// TwinCAT 3 PLC project API
// ProgramVersion: 3.1.4020.4
// libraries:
//   Tc2_MC2, * (Beckhoff Automation GmbH)
//   Tc2_Standard, * (Beckhoff Automation GmbH)
//   Tc2_System, * (Beckhoff Automation GmbH)
//   Tc3_Module, * (Beckhoff Automation GmbH)
// project tree:
//   DUTs/ ST_GenericStatus.TcDUT, ST_IO.TcDUT, ST_MachineParam.TcDUT, ST_Out.TcDUT, ST_Param.TcDUT, ST_RecipeParam.TcDUT, ST_Status.TcDUT
//   GVLs/ GVL.TcGVL
//   / PlcTask.TcTTO
//   POUs/ FB_Btn.TcPOU, FB_BtnHmiAutoResetType.TcPOU, FB_CycleAuto.TcPOU, FB_CycleInit.TcPOU, FB_CycleMain.TcPOU, FB_CycleMan.TcPOU, FB_Moteur.TcPOU, FB_Station.TcPOU, MAIN.TcPOU
// real-time tasks:
//   TASK PlcTask: cycle T#10ms, priority 20, ADS port 350
// motion (NC):
//   TASK NC-Task 1 SAF: cycle T#2ms, priority 4, ADS port 501
//   TASK NC-Task 1 SVB: cycle T#10ms, priority 8, ADS port 511
//   AXIS Axe Z (id 1)
//     OtherSettings: AllowMotionCmdToSlave=true
//     encoder EncType=1
//     drive DrvType=5
//     controller CtrType=1
//       CtrPara: PriorControlFactor=1
//         Observer: BandWidth=20
// variable links:
//   API/API Instance <-> NC-Task 1 SAF/Axes/Axe Z
//     PlcTask Inputs/GVL.axeX.NcToPlc <-> Outputs/ToPlc
//     PlcTask Outputs/GVL.axeX.PlcToNc <-> Inputs/FromPlc

CONFIGURATION API
    RESOURCE PLC ON TwinCAT3
        TASK PlcTask(INTERVAL := T#10ms, PRIORITY := 20);
        PROGRAM MAIN WITH PlcTask : MAIN;
    END_RESOURCE
END_CONFIGURATION

// ---- DUTs/ST_GenericStatus.TcDUT
TYPE ST_GenericStatus :
STRUCT
	(*-------------------------------------------------------------------------------------------------
		xuton du panel HMI
	-------------------------------------------------------------------------------------------------*)
	(*mode actif plc to HMI*)
	xModeInit					:BOOL; (*selection du mode prise origine machine type flanc*)
	

	xModeAuto				:BOOL; (*selection du mode automatique type flanc*)
	xModeMan				:BOOL; (*selection du mode manuel type flanc*)
	xModeStep				:BOOL; (*selection du mode pas à pas type flanc*)
	
	xWaitStartNextStep:BOOL;

	iNcStatus				:DINT;					(*status NC*)
	iOverride:DINT;
	(*-------------------------------------------------------------------------------------------------
		Machine global state
	-------------------------------------------------------------------------------------------------*)

	(*boReadyForPower			: BOOL;					(* Condition machine prête pour faire un power on des axes*)*)
	xInitOk:BOOL;


	xPowerOff:BOOL;(*"POWER OFF": IF motor power AND pneumatic are "OFF" (Emergency stop)*)

	xPowering:BOOL;(*"POWERING": Transition mode*)

	xPowerOn:BOOL;(*"POWER ON": Motor power "ON", pneumatic "ON"*)

	xInitializing:BOOL;(*"INITIALISING": Transition mode, INIT cycle*)

	xReady:BOOL;(*"READY": Ready FOR AUTO mode Green*)

	xRunning:BOOL;(*"RUNNING": running in AUTO mode*)

	xStoping:BOOL;(*"STOPPING": Normally stopping  in AUTO mode*)

	xReseting:BOOL;(*"RESETING": Reset cycle operation, can be DO in every situation AND mode*)

	(*Status light*)
	byStatusLight:BYTE; (*bit0=1 red light, bit1=1 red light blink, bit2=1 yelow, bit3=1 yelow blink, bit4=1 green, bit5=1 green blink*)

END_STRUCT
END_TYPE

// ---- DUTs/ST_IO.TcDUT
TYPE ST_IO :
STRUCT
	stOut: ST_Out;
END_STRUCT
END_TYPE

// ---- DUTs/ST_MachineParam.TcDUT
TYPE ST_MachineParam :
STRUCT
	
END_STRUCT
END_TYPE

// ---- DUTs/ST_Out.TcDUT
TYPE ST_Out :
STRUCT
	xMotEnable: BOOL;
	xMotPosBasse: BOOL;
	xMotPosHaute: BOOL;
END_STRUCT
END_TYPE

// ---- DUTs/ST_Param.TcDUT
TYPE ST_Param :
STRUCT
	
	(*NOVRAM (Non-Volatile Random Access Memory) persistent variables *)
	(*Parameters*)
	stStatus		:ST_Status;	(*Machine global status structure ~(OPC :1:)*)
	stMachine		:ST_MachineParam ;	(*Machine parameters structure editing from HMI ~(OPC :1:)*)
	stRecipe		:ST_RecipeParam;	(*Recipe parameters structure editing from HMI ~(OPC :1:)*)
	//stReporting		:ST_Reporting;
	

END_STRUCT
END_TYPE

// ---- DUTs/ST_RecipeParam.TcDUT
TYPE ST_RecipeParam :
STRUCT

	(*Paramètres production*)
	lrPositionBasse: LREAL;
	lrVitesse: LREAL;
	
END_STRUCT
END_TYPE

// ---- DUTs/ST_Status.TcDUT
TYPE ST_Status :
STRUCT
	(*Common*)
	stCommon:ST_GenericStatus;	(*Common*)

	(*Activation from HMI*)
	inJogSelectCylinder:INT;(**)
	inJogSelectMotor: INT;
	iNiveauUtilisateur:INT;
	sUserName:STRING[100]:='';//user name from HMI
	
	iCounterPiecesProduites: INT;                             (*Nombre de pièces produites (=nombre de pièces triées)*)
	iCounterPiecesBonnes: INT;
	iCounterPiecesMauvaises: INT;
	iCounterLaser:DINT;//compteur de cycle laser limite à 4'000'000
	diCounterError:DINT;
	//sMessageHmi: STRING(200);
	sMessageHmiStatus: STRING(50);	
	sBatchNo:STRING[50];
	
	//indique le niveau, vrai si plus gand ou égale
	xNiveau1:BOOL;
	xNiveau2:BOOL;
	xNiveau3:BOOL;
	xNiveau4:BOOL;
	
	lrPositionMoteur: LREAL;
	
END_STRUCT
END_TYPE

// ---- GVLs/GVL.TcGVL
VAR_GLOBAL
fbStation		:FB_Station;(*Function Block for  station*)
stIO: ST_IO;
axeX: AXIS_REF;
END_VAR

VAR_GLOBAL PERSISTENT
stParam:ST_Param;//Basis structure with all parameters and status
END_VAR

// ---- POUs/MAIN.TcPOU
PROGRAM MAIN
VAR
END_VAR

fbStation();

GVL.stParam.stStatus.lrPositionMoteur:=GVL.axeX.NcToPlc.ActPos;

GVL.stIO.stOut.xMotPosBasse:=GVL.axeX.NcToPlc.ActPos<=GVL.stParam.stRecipe.lrPositionBasse+0.01;

GVL.stIO.stOut.xMotPosHaute:=GVL.axeX.NcToPlc.ActPos>=-0.01;

END_PROGRAM

// ---- POUs/FB_Station.TcPOU
FUNCTION_BLOCK FB_Station
VAR_INPUT
	(*Objets*)
	
	
	(*Function block for cycle*)
	fbCycleMain:FB_CycleMain;
	fbCycleInit:FB_CycleInit;
	fbCycleMan:FB_CycleMan;
	fbCycleAuto:FB_CycleAuto;
	
	fbAxeX: FB_Moteur;
	
	
	(*Function blockfor small HMI button*)
	fbBtn:FB_Btn;	(*station Input and ouput*)

	(*Error management*)
//	fbErrorAdmin		:FB_ErrorAdmin;	(*FUNCTION block for error administration  *)
	
	
	
END_VAR
VAR_OUTPUT

END_VAR
VAR
	
END_VAR

//fbErrorAdmin.mResetIndex();
(************************************************************************************)
(*							Refresh cycle			 *)
(************************************************************************************)
ACT_Cycle();
ACT_Refresh();
//fbIO();
fbBtn();

fbCycleMain();

ACT_ActionActionneur();

ACTION ACT_ActionActionneur:
fbAxeX.fbHome.Execute:=fbStation.fbCycleInit.iStep=100;
fbAxeX.fbReset.Execute:=fbStation.fbCycleMain.iStep=820;
fbAxeX.fbMoveAbsolute.Execute:=fbStation.fbCycleAuto.iStep=200 OR fbStation.fbCycleAuto.iStep=300;
fbAxeX(fbAxe:=GVL.axeX);
fbAxeX.fbPower.Enable:=GVL.stIO.stOut.xMotEnable;
fbAxeX.fbPower.Enable_Negative:=TRUE;
fbAxeX.fbPower.Enable_Positive:=TRUE;
END_ACTION

ACTION ACT_Cycle:


(*Start cycle in mode*)
fbCycleInit.xStart:=fbStation.fbCycleMain.iStep=150;

fbCycleMan.xStart:=fbStation.fbCycleMain.iStep=200;

fbCycleAuto.xStart:=fbStation.fbCycleMain.iStep=305;
//fbCycleAuto.xStopCmdPin:=fbStation.fbCycleMain.iStep=390  OR fbStation.fbCycleMain.iStep=800;


fbCycleInit( );
fbCycleMan(  );
fbCycleAuto( );
END_ACTION

ACTION ACT_Refresh:
	


	(*"POWER OFF": IF motor power AND pneumatic are "OFF" (Emergency stop)
	IF this machine is selected AND power Off, it correspond TO an alarm. Red is OK.
	IF this machine isn't selected and power Off, it must be white.*)
	//stParam.stStatus.stCommon.xPowerOff:=fbStation.fbIO.In.IxEstopBtnOnly;

	(*"POWERING": Transition mode
	IF the machines are powering but without alarms OR warnings, they can blink in light blue.
	IF the machines are powering but with warning, they can blink in yellow.
	IF the machines are powering but with alarms, they can blink in red.*)
	stParam.stStatus.stCommon.xPowering:=FALSE;

	(*"POWER ON": Motor power "ON", pneumatic "ON"
	IF the machines are power On but without alarms OR warnings, they can be light blue.
	IF the machines are power On but with warning, they can be yellow.
	IF the machines are power On but with alarms, they can be red.*)
	//stParam.stStatus.stCommon.xPowerOn:=NOT fbStation.fbIO.In.IxEstopBtnOnly;

	(*"INITIALISING": Transition mode, INIT cycle
	IF the machines are initializing but without alarms OR warnings, they can blink in green.
	IF the machines are initializing but with warning, they can blink in yellow.
	IF the machines are initializing but with alarms, they can blink in red.*)
	stParam.stStatus.stCommon.xInitializing:=fbStation.fbCycleMain.iStep>100 AND fbStation.fbCycleMain.iStep<199;

	

	(*"RUNNING": running in AUTO mode
	IF the machines are running but without alarms OR warnings, they can blink in green.
	IF the machines are running but with warning, they can blink in yellow.
	IF the machines are running but with alarms, they can blink in red (NOT possible).*)
	stParam.stStatus.stCommon.xRunning:= fbStation.fbCycleAuto.xBusy
										OR fbStation.fbCycleInit.xBusy OR fbStation.fbCycleMan.iStep>5;
										
	stParam.stStatus.stCommon.xReady:=NOT stParam.stStatus.stCommon.xRunning
								 AND stParam.stStatus.stCommon.xPowerOn
								AND stParam.stStatus.iNiveauUtilisateur>0;
								 
	(*"STOPPING": Normally stopping  in AUTO mode
	IF the machines are stopping but without alarms OR warnings, they can blink in green.
	IF the machines are stopping but with warning, they can blink in yellow.
	IF the machines are stopping but with alarms, they can blink in red (NOT possible).*)
	stParam.stStatus.stCommon.xStoping:=fbStation.fbCycleMain.iStep=390  OR fbStation.fbCycleMain.iStep=800;

	(*"RESETING": Reset cycle operation, can be DO in every situation AND mode
	IF the machines are stopping but without alarms OR warnings, they can blink in green.
	IF the machines are stopping but with warning, they can blink in yellow.
	IF the machines are stopping but with alarms, they can blink in red.*)
	stParam.stStatus.stCommon.xReseting:=fbStation.fbCycleMain.xReseting;


IF stParam.stStatus.stCommon.xRunning
		THEN
		 IF stParam.stStatus.stCommon.xWaitStartNextStep 
			 THEN
			 	stParam.stStatus.sMessageHmiStatus:='SETP BY STEP';
			 ELSE
				stParam.stStatus.sMessageHmiStatus:='RUN';
		END_IF
		ELSE
			stParam.stStatus.sMessageHmiStatus:='READY';
END_IF

stParam.stStatus.xNiveau1:=stParam.stStatus.iNiveauUtilisateur>0;
stParam.stStatus.xNiveau2:=stParam.stStatus.iNiveauUtilisateur>1;
stParam.stStatus.xNiveau3:=stParam.stStatus.iNiveauUtilisateur>2;
stParam.stStatus.xNiveau4:=stParam.stStatus.iNiveauUtilisateur>3;

//Visibilité/invisibilité des boutons de quittance:
(*
stParam.stStatus.xBtnQuittanceBal1Visible:=	fbStation.fbCycleBalance1.iStep=802
												OR fbStation.fbCycleBalance1.iStep=842
												OR fbStation.fbCycleVerifEtatStation.iStep=160;
stParam.stStatus.xBtnQuittanceBal2Visible:=	fbStation.fbCycleBalance2.iStep=804	
												OR fbStation.fbCycleBalance2.iStep=844
												OR fbStation.fbCycleVerifEtatStation.iStep=210;
stParam.stStatus.xBtnQuittanceUsiVisible:=	fbStation.fbCycleUsinage.iStep=812
												OR fbStation.fbCycleVerifEtatStation.iStep=260;
*)
END_ACTION

END_FUNCTION_BLOCK

// ---- POUs/FB_CycleMain.TcPOU
FUNCTION_BLOCK FB_CycleMain
(**)
VAR_INPUT

END_VAR
VAR_OUTPUT
	xBusy				:BOOL;(*Busy output*)
	xReseting:BOOL;(*reseting mode*)
	xReadyForChangingMode:bool;
	xEStopOut:BOOL;
END_VAR
VAR_IN_OUT
END_VAR
VAR
	iStep			: INT:=0;		(* cycle step *)
	inOldStep			:INT:=0;
	fbTrigStart			: R_Trig;	(*Trigger for start*)
	
	xMemCycleAutoRun:BOOL;
	
	fbTimer:TON;
	fbTimerResetAuto:ton;
END_VAR



ACT_ChangingMode();


IF fbStation.fbBtn.HmiReset.xRisingEdge AND iStep<800
	THEN
		iStep:=800;
END_IF

CASE  iStep OF

	(********************************************************************************************************************************************************)
	(*Plc Start*)
	(********************************************************************************************************************************************************)
	0:	(*Init*)
		iStep:=50;
	
		
	(*Select mode*)
	50:(*Wait end of cycle man init auto*)
		//boEndOfProdPout:=FALSE;
		IF xReadyForChangingMode
			THEN
				iStep:=55;
		END_IF
		
	55:	(*Changing mode from HMI*)
		(*Select  Mode*)
		IF  stParam.stStatus.stCommon.xModeInit
			THEN
				iStep:=100; (*Init mode*)
		END_IF
		IF stParam.stStatus.stCommon.xModeMan 
			THEN
				iStep:=200; (*Manual mode*)
		END_IF
		IF stParam.stStatus.stCommon.xModeAuto
			THEN
					iStep:=300;(*Auto mode*)
		END_IF

	(************************************************************************************)
	(*							INIT mode						 *)
	(************************************************************************************)
	(*Wait for start cycle or changing mode*)
	100:
		IF NOT stParam.stStatus.stCommon.xModeInit
			THEN
				iStep:=50;(*select mode*)
			ELSE
				(*Start init*)
				IF (fbStation.fbBtn.HmiStart.xRisingEdge)
					THEN
						iStep:=150;
				END_IF
		END_IF

	150:(*Exit on normal end*)
		IF fbStation.fbCycleInit.xDone
			THEN
				iStep:=190;
		END_IF
		(*Exit on reset*);
		(*Exit with error level 2*)
	(*End of INIT mode*)
	190:
		//changement de mode automatique AUTO
		iStep:=50;

	(************************************************************************************)
	(*							MAN mode						 *)
	(************************************************************************************)
	(*changing mode*)
	200:
		IF NOT stParam.stStatus.stCommon.xModeMan 
			THEN
				(*select mode*)
				iStep:=290;
		END_IF
	290:(*	stParam.stStatus.dsMotPortiqueM1.xKillMotor:=FALSE;
		stParam.stStatus.dsMotPortiqueM2.xKillMotor:=FALSE;
		stParam.stStatus.dsMotPump.xKillMotor:=FALSE;*)
		IF NOT fbStation.fbCycleMan.xBusy
				THEN
					iStep:=50;
		END_IF
		

	(************************************************************************************)
	(*							AUTO mode						 *)
	(************************************************************************************)
	(*changing mode*)
	300:
		IF NOT stParam.stStatus.stCommon.xModeAuto
			THEN
				iStep:=50;(*select mode*)
			ELSE
				//Start cycle auto normal
				IF (fbStation.fbBtn.HmiStart.xRisingEdge)
					THEN
						iStep:=305;
				END_IF
		END_IF
	
	305: IF NOT fbStation.fbCycleAuto.xDone
		THEN
			iStep:=310;
	END_IF	
		
	(*Control*)
	310:IF fbStation.fbCycleAuto.xDone
		THEN
			GVL.stParam.stStatus.iCounterPiecesProduites:=GVL.stParam.stStatus.iCounterPiecesProduites+1;
			iStep:=300;
	END_IF

	(************************************************************************************)
	(*							Resetting mode					 *)
	(************************************************************************************)
	800:(*IF NOT fbStation.fbCycleAuto.xBusy OR fbTimerResetAuto.Q
			THEN
				iStep:=805;
		END_IF*)
		fbStation.fbCycleAuto.xReset:=TRUE;
		fbStation.fbCycleInit.xReset:=TRUE;
		fbStation.fbCycleMan.xReset:=TRUE;
		GVL.stIO.stOut.xMotEnable:=FALSE;
		iStep:=810;
		
	
	810:IF NOT fbStation.fbCycleInit.xBusy
		AND NOT fbStation.fbCycleMan.xBusy
		AND NOT fbStation.fbCycleAuto.xBusy
		THEN
			iStep:=820;
		END_IF
		
	820: IF fbStation.fbAxeX.fbReset.Done
		 THEN
		 	iStep:=830;
	END_IF
	
	830: GVL.stIO.stOut.xMotEnable:=TRUE;
		iStep:=50;

END_CASE

(********************************************************************************************************************************************************)
(*Special Interrupt*)
(********************************************************************************************************************************************************)




fbTimer(IN:=iStep=20 OR iStep=807 OR iStep=809 OR iStep=841 );
fbTimerResetAuto(IN:=iStep=800,pt:=T#1000MS);


xBusy:=(iStep<>0);
xReseting:=(iStep>799 AND iStep<900);



xReadyForChangingMode:= (iStep=100 OR iStep=200 OR iStep=300 OR iStep=50 OR iStep=55)
			AND NOT fbStation.fbCycleInit.xBusy
			AND NOT fbStation.fbCycleAuto.xBusy;

xEStopOut:= (iStep>899);


(********************************************************************************************************************************************************)
(*Status settings*)
(********************************************************************************************************************************************************)

xBusy:=(iStep<>0);
xReseting:=(iStep>799 AND iStep<900);

ACTION ACT_ChangingMode:
(*********************************************************************************)
(*			Changing mode														 *)
(*********************************************************************************)
IF (fbStation.fbBtn.Init.xRisingEdge 
	) 
	AND xReadyForChangingMode 
	THEN
		stParam.stStatus.stCommon.xModeInit:=TRUE;
		stParam.stStatus.stCommon.xModeAuto:=FALSE;
		stParam.stStatus.stCommon.xModeMan:=FALSE;
END_IF

IF fbStation.fbBtn.Auto.xRisingEdge 
	AND xReadyForChangingMode
 OR iStep=190 AND stParam.stStatus.stCommon.xInitOk
	THEN
		stParam.stStatus.stCommon.xModeInit:=FALSE;
		stParam.stStatus.stCommon.xModeAuto:=TRUE;
		stParam.stStatus.stCommon.xModeMan:=FALSE;
END_IF

IF fbStation.fbBtn.Man.xRisingEdge AND xReadyForChangingMode
	THEN
		stParam.stStatus.stCommon.xModeInit:=FALSE;
		stParam.stStatus.stCommon.xModeAuto:=TRUE;
		stParam.stStatus.stCommon.xModeMan:=FALSE;
END_IF
END_ACTION

ACTION ACT_ForceInitAllAxe:
stParam.stStatus.stCommon.xInitOk:=FALSE;
END_ACTION

END_FUNCTION_BLOCK

// ---- POUs/FB_CycleInit.TcPOU
(**********************************************************************************************************************************************************************
*{He-Arc}  {Hôtle de ville 7}   {2400 Le Locle}       Phone: ++ 0041 (0)32 930 13 13     Fax: ++ 0041 (0)32 930 13 14         Email: ingenierie@he-arc.ch
*=======================================================================================================================
* {Give the complete list of every blocks for a source file with several blocks}
*
*=======================================================================================================================
*Description: Cutting station init cycle
*
*=======================================================================================================================
*Version:        Date:               Author:                           Reason of modification:
*1.0                   27.11.11         Fabien Golay              Initial Version 
*1.1                                                                 
*
*
************************************************************************************************************************************************************************)
FUNCTION_BLOCK FB_CycleInit
(**)
VAR_INPUT
	xStart			:BOOL; (*start input command*)
	xReset			:BOOL; (*Reset input command*)
END_VAR
VAR_OUTPUT
	xDone			:BOOL;(*Done output*)
	xBusy				:BOOL;(*Busy output*)
END_VAR

VAR
	iStep			: INT;		(* cycle step *)
	fbTrigStart			: R_TRIG;	(*Trigger for start*)
	fbTimer:TON;
END_VAR

(*Reset  if xReset is set to true*)
IF xReset
	THEN
		xReset:=FALSE;
		iStep:=0;
		xDone:=FALSE;
END_IF


(********************************************************************************************************************)
(*			Start cycle																 *)
(*********************************************************************************************************************)
fbTrigStart(clk:=xStart );


CASE  iStep OF
	 (* Activation du cycle*)
	0:	IF fbTrigStart.Q
		THEN
			iStep:=50;
			xDone:=FALSE;
			stParam.stStatus.stCommon.xInitOk:=FALSE;
		END_IF

	50:	iStep:=100;
	fbStation.fbAxeX.fbHome.HomingMode:=MC_Direct;
	fbStation.fbAxeX.fbHome.Position:=0;

(********************************************************************************************************************)
(*				Init moteurs																		*)
(********************************************************************************************************************)

	(*monter les deux système de portique et fermer les iSteps*)
	100: IF fbStation.fbAxeX.fbHome.Done
		 THEN
		 	iStep:=999;
	END_IF
	
	 

(***********************************************************************************)
(*                           End of cycle                                                                                    *)
(************************************************************************************)
	999:xDone:=TRUE;
			iStep:=0;

END_CASE

(********************************************************************************************************************************************************)
(*Special Interrupt*)
(********************************************************************************************************************************************************)

fbTimer();

(********************************************************************************************************************************************************)
(*Status settings*)
(********************************************************************************************************************************************************)

xBusy:=(iStep<>0);

END_FUNCTION_BLOCK

// ---- POUs/FB_CycleMan.TcPOU
(**********************************************************************************************************************************************************************
*{He-Arc}  {Hôtle de ville 7}   {2400 Le Locle}       Phone: ++ 0041 (0)32 930 13 13     Fax: ++ 0041 (0)32 930 13 14         Email: ingenierie@he-arc.ch
*=======================================================================================================================
* {Give the complete list of every blocks for a source file with several blocks}
*
*=======================================================================================================================
*Description: Cutting station manual cycle
*
*=======================================================================================================================
*Version:        Date:               Author:                           Reason of modification:
*1.0                   27.11.11         Fabien Golay              Initial Version 
*1.1                                                                 
*
*
************************************************************************************************************************************************************************)
FUNCTION_BLOCK FB_CycleMan
(**)
VAR_INPUT
	xStart			:BOOL; (*start input command*)
	xStopCmdPin			:BOOL; (*stop input command*)
	xReset			:BOOL; (*Reset input command*)

END_VAR
VAR_OUTPUT
	xDone			:BOOL;(*Done output*)
	xBusy				:BOOL;(*Busy output*)
	xReady				:BOOL;(*Busy output*)
	iStep			: INT;		(* cycle step *)
END_VAR
VAR_IN_OUT
	//fbErrorAdmin:FB_ErrorAdmin;
END_VAR
VAR
	
	fbTrigStart			: R_Trig;	(*Trigger for start*)
	fbTimer:TON;
END_VAR

(*Reset  if xReset is set to true*)
IF xReset
	THEN
		xReset:=FALSE;
		iStep:=0;
		xDone:=FALSE;
END_IF
(********************************************************************************************************************************************************)
(*								Start Management																 *)
(********************************************************************************************************************************************************)
fbTrigStart(CLK:=xStart );

CASE  iStep OF

	(* Activation du cycle*)
	0:	IF fbTrigStart.Q  THEN
		iStep:=5;
	END_IF

	 (*Selecte action type from HMI*)
	5:
 (********************************************************************************************************************************************************)
(*Gestion des vérins																							*)
(********************************************************************************************************************************************************)
	(*Rentrée vérin*)
 END_CASE

END_FUNCTION_BLOCK

// ---- POUs/FB_CycleAuto.TcPOU
FUNCTION_BLOCK FB_CycleAuto
(**)
VAR_INPUT
	xStart			:BOOL; (*start input command*)
	//xStopCmdPin			:BOOL; (*stop input command*)
	xReset			:BOOL; (*Reset input command*)
		(*Station index*)
	
END_VAR
VAR_OUTPUT
	xDone			:BOOL;(*Done output*)
	xBusy				:BOOL;(*Busy output*)
END_VAR
VAR_IN_OUT
	//fbErrorAdmin:FB_ErrorAdmin;
END_VAR
VAR
	

	iStep			: INT;		(* cycle step *)
	iNextStep			: INT;		(* cycle step *)
	fbTrigStart			: R_Trig;	(*Trigger for start*)
	fbTimerTON			:TON;
	
END_VAR

(*Reset  if xReset is set to true*)
IF xReset
	THEN
		xReset:=FALSE;
		iStep:=0;
		xDone:=FALSE;
END_IF

fbTrigStart(CLK:=xStart);


CASE  iStep OF
	0:	IF fbTrigStart.Q
		THEN
		xDone:=FALSE;
		iStep:=100;
		END_IF
	
	100: fbStation.fbAxeX.fbMoveAbsolute.Position:=GVL.stParam.stRecipe.lrPositionBasse;
			fbStation.fbAxeX.fbMoveAbsolute.Velocity:=GVL.stParam.stRecipe.lrVitesse;
			iStep:=200;
			
	200: IF  fbStation.fbAxeX.fbMoveAbsolute.Done
		THEN
			iStep:=250;
	END_IF
	
	250:  fbStation.fbAxeX.fbMoveAbsolute.Position:=0;
			fbStation.fbAxeX.fbMoveAbsolute.Velocity:=GVL.stParam.stRecipe.lrVitesse;
			iStep:=300;
			
	300: IF  fbStation.fbAxeX.fbMoveAbsolute.Done
		THEN
			iStep:=900;
	END_IF

	900: xDone:=TRUE;
		iStep:=0;

END_CASE

fbTimerTON(IN:=iStep=210);
xBusy:=iStep<>0;

END_FUNCTION_BLOCK

// ---- POUs/FB_Moteur.TcPOU
FUNCTION_BLOCK FB_Moteur
VAR_INPUT
	fbPower: MC_power;
	fbMoveAbsolute: MC_MoveAbsolute;
	fbHome: MC_Home;
	fbReset: MC_Reset;
END_VAR
VAR_OUTPUT
END_VAR
VAR
	
END_VAR
VAR_IN_OUT
	fbAxe: AXIS_REF;
END_VAR

fbPower(Axis:=fbAxe);
fbMoveAbsolute(Axis:=fbAxe);
fbHome(Axis:=fbAxe);
fbReset(Axis:=fbAxe);

END_FUNCTION_BLOCK

// ---- POUs/FB_Btn.TcPOU
FUNCTION_BLOCK FB_Btn
VAR_INPUT
 (*exemple : Btn                                                             :FB_BtnHmiType; (**)*)

	HmiStart:			FB_BtnHmiAutoResetType; (*Start button*)
	HmiStop:			FB_BtnHmiAutoResetType; (*Stop button*)
	HmiReset:			FB_BtnHmiAutoResetType;
	ResetAllHoming:		FB_BtnHmiAutoResetType;
	Init:				FB_BtnHmiAutoResetType; (*Start button*)
	Man:				FB_BtnHmiAutoResetType; (*Stop button*)
	Auto:				FB_BtnHmiAutoResetType; (*Reset button*)
//	Step:				FB_BtnHmiAutoResetType; (*Set step by step mode*)




(************************************************************************************)
(*      Boutons du mode manuel                                                                                *)
(************************************************************************************)

END_VAR
VAR_OUTPUT
END_VAR
VAR

END_VAR

HmiStart();
HmiStop();(**)
HmiReset();(**)
ResetAllHoming();
Init();
Auto();
Man();
//Step(); (**)

END_FUNCTION_BLOCK

// ---- POUs/FB_BtnHmiAutoResetType.TcPOU
FUNCTION_BLOCK FB_BtnHmiAutoResetType
VAR_INPUT
	xEtat: BOOL;
END_VAR
VAR_OUTPUT
	xRisingEdge: BOOL;
END_VAR
VAR
	fbRTrig: R_Trig;
END_VAR

fbRTrig(CLK:=xEtat);
xRisingEdge:=fbRTrig.Q;
xEtat:=FALSE;

END_FUNCTION_BLOCK
